// Mitsubishi GX Works2 project: 22-1-10起保停在呼叫程序中的应用   PLC: FX1N/FX1NC

PROGRAM MAIN
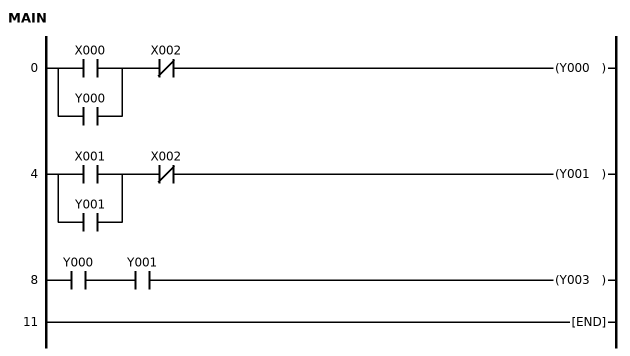
0     LD      X000
      OR      Y000
      ANI     X002
      OUT     Y000
4     LD      X001
      OR      Y001
      ANI     X002
      OUT     Y001
8     LD      Y000
      AND     Y001
      OUT     Y003
11    END
END_PROGRAM
